FUNCTION_BLOCK "FB_SortingHeightAdvanced"   // FB18, SCL
{ S7_Optimized_Access := 'FALSE' }
VERSION : 0.4
// MANTIS â€” Scene 18: Sorting by Height (Advanced)  v0.4
//  Turntable-based 2-way sort: tall items â†’ LEFT, short â†’ RIGHT.
//  DB27, 76 bytes.  Enable flag at byte 74.
// 
//  I/O from Factory I/O driver (Siemens S7-1200/1500):
//    Inputs  %I0.0â€“%I1.7  (16 BOOLs)
//    Outputs %Q0.0â€“%Q1.4  (13 BOOLs) + %QD100 (DINT counter)
// 
//  Turntable notes:
//    Turn activates CW rotation; turntable snaps to 90Â° detents on stop.
//    AtFront = TRUE when turntable faces entry conveyor (0Â° position).
//    RIGHT exit â‰ˆ 90Â° CW from front  â†’ single turn, easy.
//    LEFT  exit â‰ˆ 270Â° CW from front â†’ timer-based (TURN_LEFT_TICKS).
//    Return to FRONT: Turn ON until AtFront = TRUE (always reliable).
//  ===== SENSORS (from Factory I/O) =====
   VAR
      AtEntry : Bool;   // %I0.0 Item at entry conveyor
      LowBox : Bool;   // %I0.1 Low height sensor triggered
      HighBox : Bool;   // %I0.2 High height sensor triggered
      AtTurntableEntry : Bool;   // %I0.3 Item at turntable entry area
      AtLoadPosition : Bool;   // %I0.4 Item centred on turntable
      AtUnloadPosition : Bool;   // %I0.5 Item at turntable unload edge
      AtFront : Bool;   // %I0.6 Turntable facing front (entry)
      AtRightEntry : Bool;   // %I0.7 Item entering right conveyor
      AtLeftEntry : Bool;   // %I1.0 Item entering left conveyor
      AtRightExit : Bool;   // %I1.1 Item at right conveyor exit
      AtLeftExit : Bool;   // %I1.2 Item at left conveyor exit
      BtnStart : Bool;   // %I1.3 Start button
      BtnReset : Bool;   // %I1.4 Reset button
      BtnStop : Bool;   // %I1.5 Stop button
      EmergencyStop : Bool;   // %I1.6 Emergency stop
      BtnAuto : Bool;   // %I1.7 Auto mode ===== ACTUATORS (to Factory I/O) =====
      FeederConveyor : Bool;   // %Q0.0 Feeder conveyor
      EntryConveyor : Bool;   // %Q0.1 Entry conveyor
      LoadAct : Bool;   // %Q0.2 Turntable rollers inward (load)
      UnloadAct : Bool;   // %Q0.3 Turntable rollers outward (unload)
      TurnAct : Bool;   // %Q0.4 Turntable rotate CW
      LeftConveyor : Bool;   // %Q0.5 Left exit conveyor
      RightConveyor : Bool;   // %Q0.6 Right exit conveyor
      GreenIndicator : Bool;   // %Q0.7 Green indicator
      YellowIndicator : Bool;   // %Q1.0 Yellow indicator
      RedIndicator : Bool;   // %Q1.1 Red indicator
      StartLight : Bool;   // %Q1.2 Start button light
      ResetLight : Bool;   // %Q1.3 Reset button light
      StopLight : Bool;   // %Q1.4 Stop button light
      CounterOut : DInt;   // (DINT) %QD100 Item counter display ===== INTERNAL =====
      iState : Int;   // State machine
      ItemCount : Int;   // Internal item counter
      IsTall : Bool;   // TRUE = tall (HighBox), FALSE = short
      TurnTimer : Int;   // Timer for LEFT 270Â° CW rotation
      DwellTimer : Int;   // General-purpose delay timer
      Running : Bool;   // System running flag
      Enable : Bool := TRUE;   // ATTACK SURFACE â€” PLC never writes
   END_VAR
BEGIN
       // ===== PANEL LIGHTS =====
       #StartLight := #Running;
       #ResetLight := NOT #Running;
       #StopLight := NOT #Running;

       // ===== INDICATORS =====
       #GreenIndicator := #Running AND (#iState >= 10);
       #YellowIndicator := #Running AND (#iState >= 40) AND (#iState <= 55);
       #RedIndicator := NOT #EmergencyStop OR NOT #Enable;

       // ===== COUNTER OUTPUT =====
       #CounterOut := INT_TO_DINT(#ItemCount);

       // ===== SAFETY / ENABLE CHECK =====
       IF NOT #EmergencyStop OR NOT #Enable THEN
           #FeederConveyor := FALSE;
           #EntryConveyor := FALSE;
           #LoadAct := FALSE;
           #UnloadAct := FALSE;
           #TurnAct := FALSE;
           #LeftConveyor := FALSE;
           #RightConveyor := FALSE;
           #Running := FALSE;
           #iState := 0;
           RETURN;
       END_IF;

       // ===== START / STOP / RESET =====
       IF #BtnStart AND NOT #Running AND #EmergencyStop THEN
           #Running := TRUE;
           #iState := 10;
       END_IF;

       IF NOT #BtnStop OR NOT #EmergencyStop THEN
           #Running := FALSE;
           #FeederConveyor := FALSE;
           #EntryConveyor := FALSE;
           #LoadAct := FALSE;
           #UnloadAct := FALSE;
           #TurnAct := FALSE;
           #LeftConveyor := FALSE;
           #RightConveyor := FALSE;
           #iState := 0;
       END_IF;

       IF #BtnReset THEN
           #ItemCount := 0;
           #IsTall := FALSE;
           #iState := 0;
           #Running := FALSE;
           #FeederConveyor := FALSE;
           #EntryConveyor := FALSE;
           #LoadAct := FALSE;
           #UnloadAct := FALSE;
           #TurnAct := FALSE;
           #LeftConveyor := FALSE;
           #RightConveyor := FALSE;
       END_IF;

       IF NOT #Running THEN
           #FeederConveyor := FALSE;
           #EntryConveyor := FALSE;
           #LoadAct := FALSE;
           #UnloadAct := FALSE;
           #TurnAct := FALSE;
           #LeftConveyor := FALSE;
           #RightConveyor := FALSE;
           RETURN;
       END_IF;

       // ===== EXIT CONVEYORS ALWAYS ON WHILE RUNNING =====
       #LeftConveyor := TRUE;
       #RightConveyor := TRUE;

       // ===== DEFAULT PROCESS OUTPUTS OFF (states set what they need) =====
       #FeederConveyor := FALSE;
       #EntryConveyor := FALSE;
       #LoadAct := FALSE;
       #UnloadAct := FALSE;
       #TurnAct := FALSE;

       // ===== STATE MACHINE =====
       CASE #iState OF

           0: // IDLE â€” waiting for start
               ;

               // ---------- FEED ----------
           10: // Run feeder + entry conveyors, detect height
               #FeederConveyor := TRUE;
               #EntryConveyor := TRUE;
               // Latch height while item passes sensors
               IF #HighBox THEN
                   #IsTall := TRUE;
               ELSIF #LowBox AND NOT #HighBox THEN
                   #IsTall := FALSE;
               END_IF;
               IF #AtTurntableEntry THEN
                   #iState := 20;
               END_IF;

               // ---------- LOAD ONTO TURNTABLE ----------
           20: // Turntable rollers pull item in
               #EntryConveyor := TRUE;
               #LoadAct := TRUE;
               IF #AtLoadPosition THEN
                   #DwellTimer := 0;
                   IF #IsTall THEN
                       #iState := 50;   // turn LEFT (270Â° CW)
                   ELSE
                       #iState := 40;   // turn RIGHT (90Â° CW)
                   END_IF;
               END_IF;

               // --------- TURN RIGHT  (90Â° CW from FRONT) ---------
           40: // Turn CW while still at FRONT; stop once we leave
               IF #AtFront THEN
                   #TurnAct := TRUE;
               ELSE
                   #DwellTimer := 0;
                   #iState := 45;
               END_IF;

           45: // Settle at RIGHT position
               #DwellTimer := #DwellTimer + 1;
               IF #DwellTimer >= 10 THEN
                   #DwellTimer := 0;
                   #iState := 60;
               END_IF;

               // --------- TURN LEFT  (270Â° CW from FRONT) ---------
               // Timer-based: ~30 ticks after leaving FRONT covers ~270Â°.
               // Calibrate if turntable speed differs from default.
           50: // Start turning CW, wait to leave FRONT
               #TurnAct := TRUE;
               IF NOT #AtFront THEN
                   #TurnTimer := 0;
                   #iState := 51;
               END_IF;

           51: // Keep turning CW past RIGHT and BACK toward LEFT
               #TurnAct := TRUE;
               #TurnTimer := #TurnTimer + 1;
               IF #TurnTimer >= 30 THEN
                   #DwellTimer := 0;
                   #iState := 55;
               END_IF;

           55: // Settle at LEFT position
               #DwellTimer := #DwellTimer + 1;
               IF #DwellTimer >= 10 THEN
                   #DwellTimer := 0;
                   #iState := 60;
               END_IF;

               // --------- UNLOAD ---------
           60: // Push item off turntable onto exit conveyor
               #UnloadAct := TRUE;
               #DwellTimer := #DwellTimer + 1;
               IF (#IsTall AND #AtLeftEntry) OR (NOT #IsTall AND #AtRightEntry)
                   OR (#DwellTimer >= 50) THEN
                   #DwellTimer := 0;
                   #iState := 70;
               END_IF;

               // --------- EXIT CONVEYOR ---------
           70: // Wait for item to reach exit sensor
               #DwellTimer := #DwellTimer + 1;
               IF (#IsTall AND #AtLeftExit) OR (NOT #IsTall AND #AtRightExit)
                   OR (#DwellTimer >= 50) THEN
                   #DwellTimer := 0;
                   #iState := 80;
               END_IF;

               // --------- RETURN TO FRONT ---------
           80: // Turn CW until AtFront
               #TurnAct := TRUE;
               IF #AtFront THEN
                   #DwellTimer := 0;
                   #iState := 85;
               END_IF;

           85: // Settle at FRONT
               #DwellTimer := #DwellTimer + 1;
               IF #DwellTimer >= 10 THEN
                   #iState := 90;
               END_IF;

               // --------- COUNT AND LOOP ---------
           90: // Increment counter, reset flags, loop
               #ItemCount := #ItemCount + 1;
               #IsTall := FALSE;
               #iState := 10;

       END_CASE;
END_FUNCTION_BLOCK

FUNCTION_BLOCK "FB_SortingHeightBasic"   // FB19, SCL
{ S7_Optimized_Access := 'FALSE' }
VERSION : 0.4
// MANTIS â€” Scene 19: Sorting by Height (Basic)
//  Sort items by height: short â†’ LEFT, tall â†’ RIGHT.
//  DB28: Instance DB (non-optimized access)
// 
//  Factory I/O layout:
//    Entry conveyor feeds items onto a pallet/loading area.
//    High sensor detects tall items. Low sensor detects short items.
//    Pallet sensor detects pallet ready. Loaded confirms item loaded.
//    Short box (Low sensor only) â†’ Transfer LEFT.
//    Tall  box (High sensor)     â†’ Transfer RIGHT.
//    Left and right exit conveyors carry sorted items away.
//    Start/Stop/Reset/EmergencyStop/Auto on control panel.
//    Counter display shows items sorted.
// 
//  Driver mapping (from Factory I/O):
//    SENSORS (Inputs):
//      NOTE: Use %I10.x/%I11.x (NOT %I0.x/%I1.x) because the PLC's
//      built-in physical DI module owns %IB0 and overwrites external writes.
//      High sensor      â†’ %I10.0
//      Low sensor       â†’ %I10.1
//      Pallet sensor    â†’ %I10.2
//      Loaded           â†’ %I10.3
//      At left entry    â†’ %I10.4
//      At left exit     â†’ %I10.5
//      At right entry   â†’ %I10.6
//      At right exit    â†’ %I10.7
//      Start            â†’ %I11.0
//      Reset            â†’ %I11.1
//      Stop             â†’ %I11.2
//      Emergency stop   â†’ %I11.3
//      Auto             â†’ %I11.4
//      FACTORY I/O (Running) â†’ %I11.5
// 
//    ACTUATORS (Outputs):
//      Conveyor entry   â†’ %Q0.0
//      Load             â†’ %Q0.1
//      Unload           â†’ %Q0.2
//      Transf. left     â†’ %Q0.3
//      Transf. right    â†’ %Q0.4
//      Conveyor left    â†’ %Q0.5
//      Conveyor right   â†’ %Q0.6
//      Start light      â†’ %Q0.7
//      Reset light      â†’ %Q1.0
//      Stop light       â†’ %Q1.1
//      Counter          â†’ (DINT) %QD100
// 
//  DB28 byte layout (non-optimized):
//    Sensors:
//      0:  HighSensor     2: LowSensor      4: PalletSensor
//      6:  Loaded         8: AtLeftEntry    10: AtLeftExit
//     12:  AtRightEntry  14: AtRightExit
//     16:  BtnStart      18: BtnReset      20: BtnStop
//     22:  EmergencyStop 24: BtnAuto
//    Actuators:
//     26:  ConveyorEntry 28: Load          30: Unload
//     32:  TransfLeft    34: TransfRight
//     36:  ConveyorLeft  38: ConveyorRight
//     40:  StartLight    42: ResetLight    44: StopLight
//     46-49: Counter (DINT)
//    Internal:
//     50:  iState (INT)    52: ItemCount (INT)
//     54:  IsTall (BOOL)   56: DwellTimer (INT)
//     58:  Running (BOOL)  60: Enable (BOOL)
//    Total = 62 bytes
// 
//  Sorting logic:
//    Low sensor ON only â†’ short item â†’ transfer LEFT
//    High sensor ON     â†’ tall item  â†’ transfer RIGHT
// 
//  Vulnerability: Enable (byte 60, default TRUE) â€” read but NEVER written.
//  â”€â”€ Sensors (inputs) â”€â”€
   VAR
      HighSensor : Bool;   // byte 0 â€” %I0.0
      _p00 : Byte;
      LowSensor : Bool;   // byte 2 â€” %I0.1
      _p01 : Byte;
      PalletSensor : Bool;   // byte 4 â€” %I0.2
      _p02 : Byte;
      Loaded : Bool;   // byte 6 â€” %I0.3
      _p03 : Byte;
      AtLeftEntry : Bool;   // byte 8 â€” %I0.4
      _p04 : Byte;
      AtLeftExit : Bool;   // byte 10 â€” %I0.5
      _p05 : Byte;
      AtRightEntry : Bool;   // byte 12 â€” %I0.6
      _p06 : Byte;
      AtRightExit : Bool;   // byte 14 â€” %I0.7
      _p07 : Byte;
      BtnStart : Bool;   // byte 16 â€” %I1.0
      _p08 : Byte;
      BtnReset : Bool;   // byte 18 â€” %I1.1
      _p09 : Byte;
      BtnStop : Bool;   // byte 20 â€” %I1.2
      _p10 : Byte;
      EmergencyStop : Bool;   // byte 22 â€” %I1.3
      _p11 : Byte;
      BtnAuto : Bool;   // byte 24 â€” %I1.4
      _p12 : Byte;   // â”€â”€ Actuators (outputs) â”€â”€
      ConveyorEntry : Bool;   // byte 26 â€” %Q0.0
      _p13 : Byte;
      LoadAct : Bool;   // byte 28 â€” %Q0.1 (Load)
      _p14 : Byte;
      UnloadAct : Bool;   // byte 30 â€” %Q0.2 (Unload)
      _p15 : Byte;
      TransfLeft : Bool;   // byte 32 â€” %Q0.3
      _p16 : Byte;
      TransfRight : Bool;   // byte 34 â€” %Q0.4
      _p17 : Byte;
      ConveyorLeft : Bool;   // byte 36 â€” %Q0.5
      _p18 : Byte;
      ConveyorRight : Bool;   // byte 38 â€” %Q0.6
      _p19 : Byte;
      StartLight : Bool;   // byte 40 â€” %Q0.7
      _p20 : Byte;
      ResetLight : Bool;   // byte 42 â€” %Q1.0
      _p21 : Byte;
      StopLight : Bool;   // byte 44 â€” %Q1.1
      _p22 : Byte;
      CounterOut : DInt := 0;   // byte 46 â€” %QD100 â”€â”€ Internal state â”€â”€
      iState : Int := 0;   // byte 50
      ItemCount : Int := 0;   // byte 52
      IsTall : Bool := FALSE;   // byte 54
      _p23 : Byte;
      DwellTimer : Int := 0;   // byte 56
      Running : Bool := FALSE;   // byte 58
      _p24 : Byte;
      Enable : Bool := TRUE;   // byte 60 â€” system enable (default ON)
      _p25 : Byte;   // Total: 62 bytes
   END_VAR
BEGIN
       // â•â•â•â•â•â•â•â•â•â•â•â•â•â•â•â•â•â•â•â•â•â•â•â•â•â•â•â•â•â•â•â•â•â•â•â•â•â•â•â•â•â•â•â•â•â•â•â•â•â•â•â•
       // Safety gate: if Enable is FALSE, shut everything down
       // â•â•â•â•â•â•â•â•â•â•â•â•â•â•â•â•â•â•â•â•â•â•â•â•â•â•â•â•â•â•â•â•â•â•â•â•â•â•â•â•â•â•â•â•â•â•â•â•â•â•â•â•
       IF NOT #Enable THEN
           #Running := FALSE;
           #ConveyorEntry := FALSE;
           #LoadAct := FALSE;
           #UnloadAct := FALSE;
           #TransfLeft := FALSE;
           #TransfRight := FALSE;
           #ConveyorLeft := FALSE;
           #ConveyorRight := FALSE;
           #StartLight := FALSE;
           #StopLight := TRUE;
           #ResetLight := FALSE;
           RETURN;
       END_IF;

       // â•â•â•â•â•â•â•â•â•â•â•â•â•â•â•â•â•â•â•â•â•â•â•â•â•â•â•â•â•â•â•â•â•â•â•â•â•â•â•â•â•â•â•â•â•â•â•â•â•â•â•â•
       // Button handling
       //
       // Factory I/O button types for this scene:
       //   Start  â†’ momentary, normally OPEN   (FALSE=idle, TRUE=pressed)
       //   Stop   â†’ momentary, normally CLOSED (TRUE=idle, FALSE=pressed)
       //   Reset  â†’ momentary, normally OPEN   (FALSE=idle, TRUE=pressed)
       //   E-Stop â†’ latching,  normally CLOSED (TRUE=normal, FALSE=engaged)
       //   Auto   â†’ selector switch
       // â•â•â•â•â•â•â•â•â•â•â•â•â•â•â•â•â•â•â•â•â•â•â•â•â•â•â•â•â•â•â•â•â•â•â•â•â•â•â•â•â•â•â•â•â•â•â•â•â•â•â•â•

       // Emergency stop is NC: FALSE when engaged â†’ stop
       IF NOT #EmergencyStop THEN
           #Running := FALSE;
       END_IF;

       // Stop is NC: FALSE when pressed â†’ stop
       IF NOT #BtnStop THEN
           #Running := FALSE;
       END_IF;

       // Start is NO: TRUE when pressed â†’ start (only if E-stop and Stop OK)
       IF #BtnStart AND NOT #Running AND #EmergencyStop AND #BtnStop THEN
           #Running := TRUE;
       END_IF;

       // Auto-start: if E-stop normal AND Stop not pressed, start automatically
       IF #EmergencyStop AND #BtnStop AND NOT #BtnStart THEN
           #Running := TRUE;
       END_IF;

       IF #BtnReset THEN
           #Running := FALSE;
           #iState := 0;
           #ItemCount := 0;
           #CounterOut := 0;
           #DwellTimer := 0;
           #IsTall := FALSE;
           #ConveyorEntry := FALSE;
           #LoadAct := FALSE;
           #UnloadAct := FALSE;
           #TransfLeft := FALSE;
           #TransfRight := FALSE;
           #ResetLight := TRUE;
           #StartLight := FALSE;
           #StopLight := FALSE;
           RETURN;
       END_IF;

       // â•â•â•â•â•â•â•â•â•â•â•â•â•â•â•â•â•â•â•â•â•â•â•â•â•â•â•â•â•â•â•â•â•â•â•â•â•â•â•â•â•â•â•â•â•â•â•â•â•â•â•â•
       // Panel indicator lights
       // â•â•â•â•â•â•â•â•â•â•â•â•â•â•â•â•â•â•â•â•â•â•â•â•â•â•â•â•â•â•â•â•â•â•â•â•â•â•â•â•â•â•â•â•â•â•â•â•â•â•â•â•
       #StartLight := #Running;
       #StopLight := NOT #Running;
       #ResetLight := FALSE;

       // â•â•â•â•â•â•â•â•â•â•â•â•â•â•â•â•â•â•â•â•â•â•â•â•â•â•â•â•â•â•â•â•â•â•â•â•â•â•â•â•â•â•â•â•â•â•â•â•â•â•â•â•
       // NOT running â†’ stop all actuators
       // â•â•â•â•â•â•â•â•â•â•â•â•â•â•â•â•â•â•â•â•â•â•â•â•â•â•â•â•â•â•â•â•â•â•â•â•â•â•â•â•â•â•â•â•â•â•â•â•â•â•â•â•
       IF NOT #Running THEN
           #ConveyorEntry := FALSE;
           #LoadAct := FALSE;
           #UnloadAct := FALSE;
           #TransfLeft := FALSE;
           #TransfRight := FALSE;
           #ConveyorLeft := FALSE;
           #ConveyorRight := FALSE;
           RETURN;
       END_IF;

       // â•â•â•â•â•â•â•â•â•â•â•â•â•â•â•â•â•â•â•â•â•â•â•â•â•â•â•â•â•â•â•â•â•â•â•â•â•â•â•â•â•â•â•â•â•â•â•â•â•â•â•â•
       // RUNNING â€” exit conveyors always ON
       // â•â•â•â•â•â•â•â•â•â•â•â•â•â•â•â•â•â•â•â•â•â•â•â•â•â•â•â•â•â•â•â•â•â•â•â•â•â•â•â•â•â•â•â•â•â•â•â•â•â•â•â•
       #ConveyorLeft := TRUE;
       #ConveyorRight := TRUE;

       // â•â•â•â•â•â•â•â•â•â•â•â•â•â•â•â•â•â•â•â•â•â•â•â•â•â•â•â•â•â•â•â•â•â•â•â•â•â•â•â•â•â•â•â•â•â•â•â•â•â•â•â•
       // Sorting state machine
       //   State 0: Feed â€” run entry conveyor, latch height, wait for pallet
       //   State 1: Load â€” lift transfer chains, wait for Loaded sensor
       //   State 2: Transfer â€” shortâ†’LEFT, tallâ†’RIGHT
       //   State 3: Clear â€” keep transfer ON while item clears center
       //   State 4: Finish â€” increment counter, return to feed
       //
       // Sorting direction:
       //   Low sensor only (short box)  â†’ Transfer LEFT
       //   High sensor (tall box)       â†’ Transfer RIGHT
       //
       // DwellTimer counts PLC scan cycles (~1-2 ms each on S7-1200).
       // Factory I/O mechanisms need real-world seconds, so thresholds
       // are in the thousands.
       // â•â•â•â•â•â•â•â•â•â•â•â•â•â•â•â•â•â•â•â•â•â•â•â•â•â•â•â•â•â•â•â•â•â•â•â•â•â•â•â•â•â•â•â•â•â•â•â•â•â•â•â•
       CASE #iState OF
           0: // â”€â”€ FEED: entry conveyor ON, detect height, wait for pallet â”€â”€
               #ConveyorEntry := TRUE;
               #LoadAct := FALSE;
               #UnloadAct := FALSE;
               #TransfLeft := FALSE;
               #TransfRight := FALSE;

               // Latch height sensors AS THE BOX APPROACHES on the entry conveyor.
               // The sensors fire as the box passes through â€” we must catch them
               // here in State 0 before the conveyor stops.
               IF #HighSensor THEN
                   #IsTall := TRUE;
               ELSIF #LowSensor THEN
                   #IsTall := FALSE;
               END_IF;

               IF #PalletSensor THEN
                   #DwellTimer := 0;
                   #iState := 1;
               END_IF;

           1: // â”€â”€ LOAD: run entry conveyor until box is fully loaded, then transfer â”€â”€
               // Entry conveyor keeps running until Loaded sensor fires
               // (box is fully on the loading platform and chains are raised).
               // Only then do we stop the conveyor and proceed to transfer.
               IF #Loaded THEN
                   #ConveyorEntry := FALSE;
               ELSE
                   #ConveyorEntry := TRUE;
               END_IF;
               #LoadAct := TRUE;         // Raise chains to lift box off rollers
               #UnloadAct := FALSE;
               #TransfLeft := FALSE;
               #TransfRight := FALSE;

               // Keep latching height sensors (they may still be active)
               IF #HighSensor THEN
                   #IsTall := TRUE;
               ELSIF #LowSensor THEN
                   #IsTall := FALSE;
               END_IF;

               #DwellTimer := #DwellTimer + 1;

               IF #Loaded THEN
                   // Box confirmed on platform â€” proceed to transfer
                   #DwellTimer := 0;
                   #iState := 2;
               ELSIF #DwellTimer > 5000 THEN
                   // Timeout (~5-10 s): Loaded never triggered, proceed anyway
                   #ConveyorEntry := FALSE;
                   #DwellTimer := 0;
                   #iState := 2;
               END_IF;

           2: // â”€â”€ TRANSFER: shortâ†’LEFT, tallâ†’RIGHT â”€â”€
               // Chains must stay raised (LoadAct=TRUE) while transfer runs.
               // Use TIMER ONLY â€” do NOT check AtLeftEntry/AtRightEntry because
               // those sensors may be permanently ON from previous boxes on the
               // exit conveyors.
               #ConveyorEntry := FALSE;
               #LoadAct := TRUE;         // KEEP chains raised during transfer!
               #UnloadAct := FALSE;

               IF #IsTall THEN
                   #TransfLeft := FALSE;
                   #TransfRight := TRUE;     // Tall â†’ RIGHT
               ELSE
                   #TransfLeft := TRUE;      // Short â†’ LEFT
                   #TransfRight := FALSE;
               END_IF;

               // Run transfer for a fixed duration (~5-10 seconds)
               #DwellTimer := #DwellTimer + 1;
               IF #DwellTimer > 5000 THEN
                   #iState := 3;
                   #DwellTimer := 0;
               END_IF;

           3: // â”€â”€ CLEAR: keep transfer ON so item fully clears center, then unload â”€â”€
               #ConveyorEntry := FALSE;

               IF #DwellTimer < 1500 THEN
                   // First ~1.5-3 s: keep chains UP + transfer running to push item off center
                   #LoadAct := TRUE;     // chains still raised
                   IF #IsTall THEN
                       #TransfLeft := FALSE;
                       #TransfRight := TRUE;
                   ELSE
                       #TransfLeft := TRUE;
                       #TransfRight := FALSE;
                   END_IF;
                   #UnloadAct := FALSE;
               ELSE
                   // Then: stop transfer, UNLOAD to lower chains back down
                   #LoadAct := FALSE;
                   #TransfLeft := FALSE;
                   #TransfRight := FALSE;
                   #UnloadAct := TRUE;
               END_IF;

               #DwellTimer := #DwellTimer + 1;
               IF #DwellTimer > 3000 THEN
                   // Total ~3-6 s dwell â€” item should be fully on exit conveyor
                   #iState := 4;
                   #DwellTimer := 0;
               END_IF;

           4: // â”€â”€ FINISH: count item, reset, return to feed â”€â”€
               #ConveyorEntry := FALSE;
               #LoadAct := FALSE;
               #UnloadAct := FALSE;
               #TransfLeft := FALSE;
               #TransfRight := FALSE;

               #ItemCount := #ItemCount + 1;
               #CounterOut := INT_TO_DINT(#ItemCount);
               #IsTall := FALSE;
               #iState := 0;

           ELSE
               // Unknown state â€” safe fallback
               #ConveyorEntry := FALSE;
               #LoadAct := FALSE;
               #UnloadAct := FALSE;
               #TransfLeft := FALSE;
               #TransfRight := FALSE;
               #iState := 0;
       END_CASE;
END_FUNCTION_BLOCK

FUNCTION_BLOCK "FB_SortingStation"   // FB20, SCL
{ S7_Optimized_Access := 'FALSE' }
VERSION : 0.1
// MANTIS â€” Scene 21: Sorting Station
//  Separate green and blue items using a vision sensor.
//  DB30: I/O mapping
   VAR
      ItemAtEntry : Bool;   // 0.0
      _pad0 : Byte;
      VisionColor : Int;   // 2 (0=none, 1=green, 2=blue)
      AtDiverter : Bool;   // 4.0
      _pad1 : Byte;
      AtExitGreen : Bool;   // 6.0
      _pad2 : Byte;
      AtExitBlue : Bool;   // 8.0
      _pad3 : Byte;
      ConveyorIn : Bool;   // 10.0
      _pad4 : Byte;
      ConveyorGreen : Bool;   // 12.0
      _pad5 : Byte;
      ConveyorBlue : Bool;   // 14.0
      _pad6 : Byte;
      Diverter : Bool;   // 16.0 (FALSE=green, TRUE=blue)
      _pad7 : Byte;
      Emitter : Bool;   // 18.0
      _pad8 : Byte;
      RemoverGreen : Bool;   // 20.0
      _pad9 : Byte;
      RemoverBlue : Bool;   // 22.0
      _pad10 : Byte;
      DetectedColor : Int := 0;
   END_VAR
BEGIN
       #Emitter := TRUE;
       #ConveyorIn := TRUE;
       #ConveyorGreen := TRUE;
       #ConveyorBlue := TRUE;
       #RemoverGreen := TRUE;
       #RemoverBlue := TRUE;

       // Detect color
       IF #ItemAtEntry AND #VisionColor > 0 THEN
           #DetectedColor := #VisionColor;
       END_IF;

       // Divert based on color
       IF #AtDiverter THEN
           IF #DetectedColor = 1 THEN
               #Diverter := FALSE;  // Green path
           ELSIF #DetectedColor = 2 THEN
               #Diverter := TRUE;   // Blue path
           END_IF;
       END_IF;
END_FUNCTION_BLOCK

FUNCTION_BLOCK "FB_SortingWeight"   // FB21, SCL
{ S7_Optimized_Access := 'FALSE' }
VERSION : 1.0
// MANTIS â€” Scene 20: Sorting by Weight
//  3-way weight sorter: weigh each box, then send left / forward / right.
//  DB22: Instance DB for FB_SortingWeight (non-optimized access)
// 
//  Factory I/O connections (ComDrvS7):
//    INPUTS (Bool Inputs Offset=10):
//      At scale entry  â†’ %I10.0      At forward entry â†’ %I10.5
//      At scale        â†’ %I10.1      At exit front    â†’ %I10.6
//      At scale exit   â†’ %I10.2      At right entry   â†’ %I10.7
//      At left entry   â†’ %I10.3      At exit right    â†’ %I11.0
//      At exit left    â†’ %I10.4      Start            â†’ %I11.1
//                                    Reset            â†’ %I11.2
//                                    Stop             â†’ %I11.3
//                                    Auto             â†’ %I11.4
//                                    FIO Running      â†’ %I11.5
//      Weight          â†’ %ID100 (REAL)
// 
//    OUTPUTS (Bool Outputs Offset=0):
//      Entry conveyor  â†’ %Q0.0       Front conveyor   â†’ %Q0.7
//      Load scale      â†’ %Q0.1       Start light      â†’ %Q1.0
//      Send left       â†’ %Q0.2       Reset light      â†’ %Q1.1
//      Left conveyor   â†’ %Q0.3       Stop light       â†’ %Q1.2
//      Send right      â†’ %Q0.4       Left count       â†’ %QD100 (DINT)
//      Right conveyor  â†’ %Q0.5       Forward count    â†’ %QD104 (DINT)
//      Send forward    â†’ %Q0.6       Right count      â†’ %QD108 (DINT)
//                                    Weight (display) â†’ %QD112 (DINT)
// 
//  DB22 byte layout (non-optimized):
//    -- Inputs --
//    Byte 0    : AtScaleEntry   (BOOL)
//    Byte 2    : AtScale        (BOOL)
//    Byte 4    : AtScaleExit    (BOOL)
//    Byte 6    : AtLeftEntry    (BOOL)
//    Byte 8    : AtExitLeft     (BOOL)
//    Byte 10   : AtForwardEntry (BOOL)
//    Byte 12   : AtExitFront    (BOOL)
//    Byte 14   : AtRightEntry   (BOOL)
//    Byte 16   : AtExitRight    (BOOL)
//    Byte 18   : BtnStart       (BOOL)
//    Byte 20   : BtnReset       (BOOL)
//    Byte 22   : BtnStop        (BOOL)
//    Byte 24   : BtnAuto        (BOOL)
//    Byte 26   : FIO_Running    (BOOL)
//    Byte 28   : Weight         (REAL)  â€” analog scale reading
//    -- Outputs --
//    Byte 32   : EntryConveyor  (BOOL)
//    Byte 34   : LoadScale      (BOOL)
//    Byte 36   : SendLeft       (BOOL)
//    Byte 38   : LeftConveyor   (BOOL)
//    Byte 40   : SendRight      (BOOL)
//    Byte 42   : RightConveyor  (BOOL)
//    Byte 44   : SendForward    (BOOL)
//    Byte 46   : FrontConveyor  (BOOL)
//    Byte 48   : StartLight     (BOOL)
//    Byte 50   : ResetLight     (BOOL)
//    Byte 52   : StopLight      (BOOL)
//    Byte 54   : LeftCount      (DINT)
//    Byte 58   : ForwardCount   (DINT)
//    Byte 62   : RightCount     (DINT)
//    Byte 66   : WeightDisplay  (DINT)
//    -- Internal --
//    Byte 70   : MeasuredWeight (REAL)
//    Byte 74   : LightThresh    (REAL)  â€” below = left
//    Byte 78   : HeavyThresh    (REAL)  â€” above = right, between = forward
//    Byte 82   : iState         (INT)
//    Byte 84   : Enable         (BOOL)
//    Total = 86 bytes
//  -- Inputs (sensors) --
   VAR
      AtScaleEntry : Bool;   // 0
      _p00 : Byte;
      AtScale : Bool;   // 2
      _p01 : Byte;
      AtScaleExit : Bool;   // 4
      _p02 : Byte;
      AtLeftEntry : Bool;   // 6
      _p03 : Byte;
      AtExitLeft : Bool;   // 8
      _p04 : Byte;
      AtForwardEntry : Bool;   // 10
      _p05 : Byte;
      AtExitFront : Bool;   // 12
      _p06 : Byte;
      AtRightEntry : Bool;   // 14
      _p07 : Byte;
      AtExitRight : Bool;   // 16
      _p08 : Byte;
      BtnStart : Bool;   // 18
      _p09 : Byte;
      BtnReset : Bool;   // 20
      _p10 : Byte;
      BtnStop : Bool;   // 22
      _p11 : Byte;
      BtnAuto : Bool;   // 24
      _p12 : Byte;
      FIO_Running : Bool;   // 26
      _p13 : Byte;
      Weight : Real;   // 28 â€” analog scale reading -- Outputs (actuators) --
      EntryConveyor : Bool;   // 32
      _p14 : Byte;
      LoadScale : Bool;   // 34
      _p15 : Byte;
      SendLeft : Bool;   // 36
      _p16 : Byte;
      LeftConveyor : Bool;   // 38
      _p17 : Byte;
      SendRight : Bool;   // 40
      _p18 : Byte;
      RightConveyor : Bool;   // 42
      _p19 : Byte;
      SendForward : Bool;   // 44
      _p20 : Byte;
      FrontConveyor : Bool;   // 46
      _p21 : Byte;
      StartLight : Bool;   // 48
      _p22 : Byte;
      ResetLight : Bool;   // 50
      _p23 : Byte;
      StopLight : Bool;   // 52
      _p24 : Byte;
      LeftCount : DInt;   // 54
      ForwardCount : DInt;   // 58
      RightCount : DInt;   // 62
      WeightDisplay : DInt;   // 66 -- Internal --
      MeasuredWeight : Real := 0.0;   // 70
      LightThresh : Real := 2.0;   // 74 â€” below this = light â†’ left
      HeavyThresh : Real := 5.0;   // 78 â€” above this = heavy â†’ right
      iState : Int := 0;   // 82
      Enable : Bool := TRUE;   // 84
      _p25 : Byte;   // 85 Total DB size: 86 bytes
   END_VAR
BEGIN
       // Exit conveyors always run to clear sorted boxes
       #LeftConveyor := TRUE;
       #FrontConveyor := TRUE;
       #RightConveyor := TRUE;

       // Lights mirror buttons
       #StartLight := #BtnStart OR #BtnAuto;
       #StopLight := #BtnStop;
       #ResetLight := #BtnReset;

       // Display current weight as integer (Ã—100 for display)
       #WeightDisplay := REAL_TO_DINT(#Weight * 100.0);

       // Default thresholds
       IF #LightThresh < 0.1 THEN
           #LightThresh := 2.0;
       END_IF;
       IF #HeavyThresh < 0.1 THEN
           #HeavyThresh := 5.0;
       END_IF;

       IF NOT #FIO_Running OR NOT #Enable THEN
           // Safe state
           #EntryConveyor := FALSE;
           #LoadScale := FALSE;
           #SendLeft := FALSE;
           #SendRight := FALSE;
           #SendForward := FALSE;
           #iState := 0;
       ELSE
           CASE #iState OF
               0: // Idle â€” feed box onto scale
                   #EntryConveyor := TRUE;
                   #LoadScale := TRUE;
                   #SendLeft := FALSE;
                   #SendRight := FALSE;
                   #SendForward := FALSE;
                   IF #AtScale THEN
                       // Box is on scale â€” stop to weigh
                       #EntryConveyor := FALSE;
                       #LoadScale := FALSE;
                       #MeasuredWeight := #Weight;
                       #iState := 1;
                   END_IF;

               1: // Weighed â€” decide direction
                   #EntryConveyor := FALSE;
                   #LoadScale := FALSE;
                   IF #MeasuredWeight < #LightThresh THEN
                       // Light â†’ send left
                       #SendLeft := TRUE;
                       #iState := 2;
                   ELSIF #MeasuredWeight >= #HeavyThresh THEN
                       // Heavy â†’ send right
                       #SendRight := TRUE;
                       #iState := 4;
                   ELSE
                       // Medium â†’ send forward
                       #SendForward := TRUE;
                       #iState := 6;
                   END_IF;

               2: // Sending left â€” wait for box to reach left entry
                   #SendLeft := TRUE;
                   #LoadScale := TRUE;  // run scale belt to push box off
                   IF #AtLeftEntry THEN
                       #SendLeft := FALSE;
                       #LoadScale := FALSE;
                       #LeftCount := #LeftCount + 1;
                       #iState := 0;
                   END_IF;

               3: // (unused â€” reserved)
                   #iState := 0;

               4: // Sending right â€” wait for box to reach right entry
                   #SendRight := TRUE;
                   #LoadScale := TRUE;
                   IF #AtRightEntry THEN
                       #SendRight := FALSE;
                       #LoadScale := FALSE;
                       #RightCount := #RightCount + 1;
                       #iState := 0;
                   END_IF;

               5: // (unused â€” reserved)
                   #iState := 0;

               6: // Sending forward â€” wait for box to reach forward entry
                   #SendForward := TRUE;
                   #LoadScale := TRUE;
                   IF #AtForwardEntry THEN
                       #SendForward := FALSE;
                       #LoadScale := FALSE;
                       #ForwardCount := #ForwardCount + 1;
                       #iState := 0;
                   END_IF;

               7: // (unused â€” reserved)
                   #iState := 0;
           END_CASE;
       END_IF;
END_FUNCTION_BLOCK

FUNCTION_BLOCK "FB_Warehouse"   // FB22, SCL
{ S7_Optimized_Access := 'FALSE' }
VERSION : 0.1
// MANTIS â€” Scene 7: Automated Warehouse
//  Transport, store and retrieve boxes from a rack using a stacker crane.
//  DB16: I/O mapping
   VAR
      AtEntry : Bool;   // 0.0
      _pad0 : Byte;
      AtExit : Bool;   // 2.0
      _pad1 : Byte;
      CraneX : Real;   // 4
      CraneZ : Real;   // 8
      CraneFork : Bool;   // 12.0
      _pad2 : Byte;
      ConveyorIn : Bool;   // 14.0
      _pad3 : Byte;
      ConveyorOut : Bool;   // 16.0
      _pad4 : Byte;
      CraneMoveX : Real;   // 18
      CraneMoveZ : Real;   // 22
      ForkExtend : Bool;   // 26.0
      _pad5 : Byte;
      ForkRetract : Bool;   // 28.0
      _pad6 : Byte;
      Emitter : Bool;   // 30.0
      _pad7 : Byte;
      TargetSlot : Int;   // 32
      iState : Int := 0;
      CurrentSlot : Int := 0;
      SLOT_SPACING_X : Real := 200.0;
      SLOT_SPACING_Z : Real := 150.0;
      COLS : Int := 5;
      TOLERANCE : Real := 15.0;
   END_VAR
BEGIN
       CASE #iState OF
           0: // Wait for box at entry
               #ConveyorIn := TRUE;
               #Emitter := TRUE;
               IF #AtEntry THEN
                   #ConveyorIn := FALSE;
                   #Emitter := FALSE;
                   // Calculate target position from slot
                   #CraneMoveX := INT_TO_REAL(#TargetSlot MOD #COLS) * #SLOT_SPACING_X;
                   #CraneMoveZ := INT_TO_REAL(#TargetSlot / #COLS) * #SLOT_SPACING_Z;
                   #iState := 1;
               END_IF;

           1: // Pick box at entry
               #ForkExtend := TRUE;
               IF #CraneFork THEN
                   #ForkExtend := FALSE;
                   #iState := 2;
               END_IF;

           2: // Move crane to target slot
               IF ABS(#CraneX - #CraneMoveX) < #TOLERANCE AND ABS(#CraneZ - #CraneMoveZ) < #TOLERANCE THEN
                   #iState := 3;
               END_IF;

           3: // Place box in slot
               #ForkRetract := TRUE;
               IF NOT #CraneFork THEN
                   #ForkRetract := FALSE;
                   // Move to next slot
                   #CurrentSlot := #CurrentSlot + 1;
                   IF #CurrentSlot > 24 THEN
                       #CurrentSlot := 0;
                   END_IF;
                   #TargetSlot := #CurrentSlot;
                   #CraneMoveX := 0.0;
                   #CraneMoveZ := 0.0;
                   #iState := 0;
               END_IF;
       END_CASE;
END_FUNCTION_BLOCK

ORGANIZATION_BLOCK "Main"   // OB1, SCL, ProgramCycle
{ S7_Optimized_Access := 'TRUE' }
VERSION : 0.1
// =============================================================================
//  MANTIS â€” TIA Portal Main Program (OB1)
//  
//  Calls the active scene's function block each scan cycle.
//  Set "ActiveScene" in DB1 to select which scene runs.
// 
//  Scene IDs:
//    1  = From A to B               (DB3)
//    2  = From A to B (Set/Reset)   (DB4)
//    3  = Filling Tank (Timers)     (DB5)
//    4  = Queue of Items (Counters) (DB6)
//    5  = Assembler                 (DB7)
//    6  = Assembler (Analog)        (DB8)
//    7  = Automated Warehouse       (DB9)
//    8  = Buffer Station            (DB10)
//    9  = Converge Station          (DB11)
//    10 = Elevator (Advanced)       (DB12)
//    11 = Elevator (Basic)          (DB13)
//    12 = Level Control             (DB14)
//    13 = Palletizer                (DB15)
//    14 = Pick & Place (Basic)      (DB16)
//    15 = Pick & Place XYZ          (DB17)
//    16 = Production Line           (DB18)
//    17 = Separating Station        (DB19)
//    18 = Sorting Height (Advanced) (DB20)
//    19 = Sorting Height (Basic)    (DB21)
//    20 = Sorting by Weight         (DB22)
//    21 = Sorting Station           (DB23)
//  =============================================================================
   VAR_INPUT
      Initial_Call : Bool;   // Initial call of this OB
      Remanence : Bool;   // =True, if remanent data are available
   END_VAR
BEGIN
       // Call the active scene FB based on DB1.ActiveScene
       // Each scene uses its own instance DB

       // ================================================================
       // I/O BRIDGE â€” Maps Factory I/O %I/%Q to Scene DB variables.
       //
       // Factory I/O communicates via physical I/O addresses (%I, %Q).
       // MANTIS reads/writes via Data Blocks (DB) using Snap7.
       // This bridge copies:
       //   %I (sensors)   â†’ DB  (before FB call)
       //   DB (actuators) â†’ %Q  (after FB call)
       //
       // I/O assignment rule:
       //   BOOL sensors:   %I10.0, %I10.1, ... (offset 10 â€” avoids S7-1200 built-in DI at %IB0)
       //   BOOL actuators: %Q0.0,  %Q0.1,  ... (sequential bits, no conflict)
       //   DWORD inputs:   %ID100, %ID104, ...
       //   DWORD outputs:  %QD100, %QD104, ...
       //
       // IMPORTANT: The S7-1200 CPU has a built-in physical digital input module
       // at %I0.0-%I0.7 (and possibly %I1.x). The PLC overwrites these from the
       // hardware pins every scan cycle, so Factory I/O PUT/GET writes to %I0.x
       // are immediately lost. ALL sensor inputs are therefore mapped to %I10.x+
       // where no physical module exists, allowing Factory I/O writes to persist.
       //
       // In the Factory I/O S7 COMM driver, set Bool Inputs Offset = 10.
       // ================================================================

       // â”€â”€ Clear ALL outputs before scene-specific writes â”€â”€
       // Prevents stale bits from a previously-active scene confusing Factory I/O.
       "Tag__639094559022291825" := 0;
       "Tag__639094559022387271" := 0;
       "Tag__639094559022442425" := 0;
       "Tag__639094559022502581" := 0;
       "Tag__639094376040963045" := 0;
       "Tag__639094376042315926" := 0;
       "Tag__639094376042397245" := 0;
       "Tag__639094376042397246" := 0;

       CASE "DB_Config".ActiveScene OF

           1:  // Scene 1: From A to B (DB3)
               // Sensors: 1 BOOL â€” remapped to %I10.x (avoid built-in DI module)
               "FB_FromAtoB_DB".Sensor := "Tag__639094376038885860";
               // Run FB
               "FB_FromAtoB_DB"();
               // Actuators: 1 BOOL (conveyor only, emitter/remover are automatic)
               "Tag__639094376037924724" := "FB_FromAtoB_DB".Conveyor;

           2:  // Scene 2: From A to B Set/Reset (DB4)
               // 3 Bool inputs remapped to %I10.x
               "FB_FromAtoB_SR_DB".SensorA := "Tag__639094376038885860";
               "FB_FromAtoB_SR_DB".SensorB := "Tag__639094376038885861";
               "FB_FromAtoB_SR_DB".FIO_Running := "Tag__639094376039046363";
               // Run FB
               "FB_FromAtoB_SR_DB"();
               // 1 Bool output: Conveyor=%Q0.0
               "Tag__639094376037924724" := "FB_FromAtoB_SR_DB".Conveyor;

           3:  // Scene 3: Filling Tank (DB5)
               // 3 Bool inputs: Fill=%I10.0, Discharge=%I10.1, FIO_Running=%I10.2
               "FB_FillingTank_DB".SensorFill := "Tag__639094376038885860";
               "FB_FillingTank_DB".SensorDrain := "Tag__639094376038885861";
               "FB_FillingTank_DB".FIO_Running := "Tag__639094376039046363";
               "FB_FillingTank_DB"();
               // 4 Bool outputs: FillValve=%Q0.0, Filling=%Q0.1, DrainValve=%Q0.2, Discharging=%Q0.3
               "Tag__639094376037924724" := "FB_FillingTank_DB".FillValve;
               "Tag__639094376038085904" := "FB_FillingTank_DB".Filling;
               "Tag__639094376038085905" := "FB_FillingTank_DB".DrainValve;
               "Tag__639094376038405653" := "FB_FillingTank_DB".Discharging;

           4:  // Scene 4: Queue of Items (DB6)
               // Sensors â€” remapped to %I10.x (avoid built-in DI module)
               "FB_QueueItems_DB".AtEntry := "Tag__639094376038885860";
               "FB_QueueItems_DB".AtExit := "Tag__639094376038885861";
               "FB_QueueItems_DB"();
               "Tag__639094376037924724" := "FB_QueueItems_DB".Conveyor;
               "Tag__639094376038085904" := "FB_QueueItems_DB".Emitter;
               "Tag__639094376038085905" := "FB_QueueItems_DB".Remover;

           5:  // Scene 5: Assembler (DB7)
               // Sensors â€” remapped to %I10.x (avoid built-in DI module)
               "FB_Assembler_DB".PartAtPickup := "Tag__639094376038885860";
               "FB_Assembler_DB".PartAtPlace := "Tag__639094376038885861";
               "FB_Assembler_DB".LidAtPickup := "Tag__639094376039046363";
               "FB_Assembler_DB".ClampSensor := "Tag__639094376039046364";
               "FB_Assembler_DB".MovingX := "Tag__639094376039046365";
               "FB_Assembler_DB".MovingZ := "Tag__639094376039205258";
               "FB_Assembler_DB"();
               "Tag__639094376037924724" := "FB_Assembler_DB".ConveyorBase;
               "Tag__639094376038085904" := "FB_Assembler_DB".ConveyorLid;
               "Tag__639094376038085905" := "FB_Assembler_DB".ConveyorOut;
               "Tag__639094376038405653" := "FB_Assembler_DB".MoveX;
               "Tag__639094376038565707" := "FB_Assembler_DB".MoveZ;
               "Tag__639094376038565708" := "FB_Assembler_DB".Clamp;
               "Tag__639094376038565709" := "FB_Assembler_DB".Emitter;

           6:  // Scene 6: Assembler Analog (DB8) â€” has REAL I/O
               // Sensors â€” remapped to %I10.x (avoid built-in DI module)
               "FB_AssemblerAnalog_DB".PartAtPickup := "Tag__639094376038885860";
               "FB_AssemblerAnalog_DB".PartAtPlace := "Tag__639094376038885861";
               "FB_AssemblerAnalog_DB".LidAtPickup := "Tag__639094376039046363";
               "FB_AssemblerAnalog_DB".ClampSensor := "Tag__639094376039046364";
               "FB_AssemblerAnalog_DB"();
               "Tag__639094376037924724" := "FB_AssemblerAnalog_DB".ConveyorBase;
               "Tag__639094376038085904" := "FB_AssemblerAnalog_DB".ConveyorLid;
               "Tag__639094376038085905" := "FB_AssemblerAnalog_DB".ConveyorOut;
               "Tag__639094376038405653" := "FB_AssemblerAnalog_DB".Clamp;
               "Tag__639094376038565707" := "FB_AssemblerAnalog_DB".Emitter;
               // NOTE: REAL I/O (PosX, PosZ, SetpointX, SetpointZ) need
               // analog mapping â€” configure in Factory I/O driver.

           7:  // Scene 7: Automated Warehouse (DB9)
               // Sensors â€” remapped to %I10.x (avoid built-in DI module)
               "FB_Warehouse_DB".AtEntry := "Tag__639094376038885860";
               "FB_Warehouse_DB".AtExit := "Tag__639094376038885861";
               "FB_Warehouse_DB".CraneFork := "Tag__639094376039046363";
               "FB_Warehouse_DB"();
               "Tag__639094376037924724" := "FB_Warehouse_DB".ConveyorIn;
               "Tag__639094376038085904" := "FB_Warehouse_DB".ConveyorOut;
               "Tag__639094376038085905" := "FB_Warehouse_DB".ForkExtend;
               "Tag__639094376038405653" := "FB_Warehouse_DB".ForkRetract;
               "Tag__639094376038565707" := "FB_Warehouse_DB".Emitter;
               // NOTE: REAL I/O (CraneX, CraneZ, CraneMoveX, CraneMoveZ) need
               // analog mapping â€” configure in Factory I/O driver.

           8:  // Scene 8: Buffer Station (DB10)
               // Sensors â€” remapped to %I10.x (avoid built-in DI module)
               "FB_BufferStation_DB".Sensor1 := "Tag__639094376038885860";
               "FB_BufferStation_DB".Sensor2 := "Tag__639094376038885861";
               "FB_BufferStation_DB".Sensor3 := "Tag__639094376039046363";
               "FB_BufferStation_DB".Sensor4 := "Tag__639094376039046364";
               "FB_BufferStation_DB".Sensor5 := "Tag__639094376039046365";
               "FB_BufferStation_DB".AtExit := "Tag__639094376039205258";
               "FB_BufferStation_DB"();
               "Tag__639094376037924724" := "FB_BufferStation_DB".Conveyor;
               "Tag__639094376038085904" := "FB_BufferStation_DB".Stopper1;
               "Tag__639094376038085905" := "FB_BufferStation_DB".Stopper2;
               "Tag__639094376038405653" := "FB_BufferStation_DB".Emitter;
               "Tag__639094376038565707" := "FB_BufferStation_DB".Remover;

           9:  // Scene 9: Converge Station (DB11)
               // Sensors â€” remapped to %I10.x (avoid built-in DI module)
               "FB_ConvergeStation_DB".SensorLeft := "Tag__639094376038885860";
               "FB_ConvergeStation_DB".SensorRight := "Tag__639094376038885861";
               "FB_ConvergeStation_DB".SensorMerge := "Tag__639094376039046363";
               "FB_ConvergeStation_DB".AtExit := "Tag__639094376039046364";
               "FB_ConvergeStation_DB"();
               "Tag__639094376037924724" := "FB_ConvergeStation_DB".ConveyorLeft;
               "Tag__639094376038085904" := "FB_ConvergeStation_DB".ConveyorRight;
               "Tag__639094376038085905" := "FB_ConvergeStation_DB".ConveyorOut;
               "Tag__639094376038405653" := "FB_ConvergeStation_DB".Emitter1;
               "Tag__639094376038565707" := "FB_ConvergeStation_DB".Emitter2;
               "Tag__639094376038565708" := "FB_ConvergeStation_DB".Remover;

           10: // Scene 10: Elevator Advanced (DB12) â€” 20 inputs, 26 BOOL + 1 DINT outputs
               // â”€â”€ Sensors (inputs) â”€â”€ NOTE: remapped to %I10.x+ to avoid built-in DI conflict
               "FB_ElevatorAdvanced_DB".At1 := "Tag__639094376038885860";
               "FB_ElevatorAdvanced_DB".At2 := "Tag__639094376038885861";
               "FB_ElevatorAdvanced_DB".At3 := "Tag__639094376039046363";
               "FB_ElevatorAdvanced_DB".AtElevator := "Tag__639094376039046364";
               "FB_ElevatorAdvanced_DB".AtEntry := "Tag__639094376039046365";
               "FB_ElevatorAdvanced_DB".AtExit := "Tag__639094376039205258";
               "FB_ElevatorAdvanced_DB".At0Low := "Tag__639094376039205259";
               "FB_ElevatorAdvanced_DB".At0High := "Tag__639094376039205260";
               "FB_ElevatorAdvanced_DB".At1Low := "Tag__639094376039365268";
               "FB_ElevatorAdvanced_DB".At1High := "Tag__639094376039365269";
               "FB_ElevatorAdvanced_DB".At2Low := "Tag__639094376039365270";
               "FB_ElevatorAdvanced_DB".At2High := "Tag__639094376039525211";
               "FB_ElevatorAdvanced_DB".At3Low := "Tag__639094376039525212";
               "FB_ElevatorAdvanced_DB".At3High := "Tag__639094376039525213";
               "FB_ElevatorAdvanced_DB".BtnStart := "Tag__639094376039685481";
               "FB_ElevatorAdvanced_DB".BtnReset := "Tag__639094376039685482";
               "FB_ElevatorAdvanced_DB".BtnStop := "Tag__639094376039685483";
               "FB_ElevatorAdvanced_DB".EmergencyStop := "Tag__639094376039846408";
               "FB_ElevatorAdvanced_DB".BtnAuto := "Tag__639094376039846409";

               "FB_ElevatorAdvanced_DB"();

               // â”€â”€ Actuators (outputs) â”€â”€
               "Tag__639094376037924724" := "FB_ElevatorAdvanced_DB".Conveyor0;
               "Tag__639094376038085904" := "FB_ElevatorAdvanced_DB".Conveyor1;
               "Tag__639094376038085905" := "FB_ElevatorAdvanced_DB".Conveyor2;
               "Tag__639094376038405653" := "FB_ElevatorAdvanced_DB".Conveyor3;
               "Tag__639094376038565707" := "FB_ElevatorAdvanced_DB".ExitConveyor;
               "Tag__639094376038565708" := "FB_ElevatorAdvanced_DB".Load;
               "Tag__639094376039846410" := "FB_ElevatorAdvanced_DB".Unload;
               "Tag__639094376040005546" := "FB_ElevatorAdvanced_DB".Up;
               "Tag__639094376038565709" := "FB_ElevatorAdvanced_DB".Down;
               "Tag__639094376040005547" := "FB_ElevatorAdvanced_DB".Slow;
               "Tag__639094376040005548" := "FB_ElevatorAdvanced_DB".WarningLight;
               "Tag__639094376040163908" := "FB_ElevatorAdvanced_DB".StartLight;
               "Tag__639094376040163909" := "FB_ElevatorAdvanced_DB".ResetLight;
               "Tag__639094376040163910" := "FB_ElevatorAdvanced_DB".StopLight;
               "Tag__639094376040323143" := "FB_ElevatorAdvanced_DB".Floor1Ind;
               "Tag__639094376040323144" := "FB_ElevatorAdvanced_DB".Floor2Ind;
               "Tag__639094376040323145" := "FB_ElevatorAdvanced_DB".Floor3Ind;
               "Tag__639094376040483081" := "FB_ElevatorAdvanced_DB".Green1;
               "Tag__639094376040483082" := "FB_ElevatorAdvanced_DB".Yellow1;
               "Tag__639094376040483083" := "FB_ElevatorAdvanced_DB".Red1;
               "Tag__639094376040642647" := "FB_ElevatorAdvanced_DB".Green2;
               "Tag__639094376040642648" := "FB_ElevatorAdvanced_DB".Yellow2;
               "Tag__639094376040642649" := "FB_ElevatorAdvanced_DB".Red2;
               "Tag__639094376040802767" := "FB_ElevatorAdvanced_DB".Green3;
               "Tag__639094376040802768" := "FB_ElevatorAdvanced_DB".Yellow3;
               "Tag__639094376040802769" := "FB_ElevatorAdvanced_DB".Red3;
               // DINT output for display
               "Tag__639094376040963045" := DINT_TO_DWORD("FB_ElevatorAdvanced_DB".Display);

           11: // Scene 11: Elevator Basic (DB13) â€” 30 inputs, 29 outputs
               // â”€â”€ Sensors (inputs) â”€â”€
               // NOTE: Use %I10.x-%I13.x to avoid built-in DI module conflict
               "FB_ElevatorBasic_DB".AtEntry := "Tag__639094376038885860";
               "FB_ElevatorBasic_DB".AtEntryLeft := "Tag__639094376038885861";
               "FB_ElevatorBasic_DB".AtExitLeft := "Tag__639094376039046363";
               "FB_ElevatorBasic_DB".AtEntry0 := "Tag__639094376039046364";
               "FB_ElevatorBasic_DB".AtExit0 := "Tag__639094376039046365";
               "FB_ElevatorBasic_DB".AtEntryRight := "Tag__639094376039205258";
               "FB_ElevatorBasic_DB".AtExitRight := "Tag__639094376039205259";
               "FB_ElevatorBasic_DB".AtExit := "Tag__639094376039205260";
               "FB_ElevatorBasic_DB".AtEntry1 := "Tag__639094376039365268";
               "FB_ElevatorBasic_DB".AtExit1 := "Tag__639094376039365269";
               "FB_ElevatorBasic_DB".AtEntry2 := "Tag__639094376039365270";
               "FB_ElevatorBasic_DB".AtExit2 := "Tag__639094376039525211";
               "FB_ElevatorBasic_DB".AtLeftLow0 := "Tag__639094376039525212";
               "FB_ElevatorBasic_DB".AtLeftHigh0 := "Tag__639094376039525213";
               "FB_ElevatorBasic_DB".AtLeftLow1 := "Tag__639094376039685481";
               "FB_ElevatorBasic_DB".AtLeftHigh1 := "Tag__639094376039685482";
               "FB_ElevatorBasic_DB".AtLeftLow2 := "Tag__639094376039685483";
               "FB_ElevatorBasic_DB".AtLeftHigh2 := "Tag__639094376039846408";
               "FB_ElevatorBasic_DB".AtRightLow0 := "Tag__639094376039846409";
               "FB_ElevatorBasic_DB".AtRightHigh0 := "Tag__639094376041124518";
               "FB_ElevatorBasic_DB".AtRightLow1 := "Tag__639094376041124519";
               "FB_ElevatorBasic_DB".AtRightHigh1 := "Tag__639094376041283188";
               "FB_ElevatorBasic_DB".AtRightLow2 := "Tag__639094376041283189";
               "FB_ElevatorBasic_DB".AtRightHigh2 := "Tag__639094376041283190";
               "FB_ElevatorBasic_DB".BtnStart := "Tag__639094376041442043";
               "FB_ElevatorBasic_DB".BtnReset := "Tag__639094376041442044";
               "FB_ElevatorBasic_DB".BtnStop := "Tag__639094376041600752";
               "FB_ElevatorBasic_DB".EmergencyStop := "Tag__639094376041600753";
               "FB_ElevatorBasic_DB".BtnAuto := "Tag__639094376041600754";

               "FB_ElevatorBasic_DB"();

               // â”€â”€ Actuators (outputs) â”€â”€
               "Tag__639094376037924724" := "FB_ElevatorBasic_DB".EntryConveyor;
               "Tag__639094376038085904" := "FB_ElevatorBasic_DB".UnloadLeft;
               "Tag__639094376038085905" := "FB_ElevatorBasic_DB".LoadLeft;
               "Tag__639094376038405653" := "FB_ElevatorBasic_DB".Conveyor0;
               "Tag__639094376038565707" := "FB_ElevatorBasic_DB".UnloadRight;
               "Tag__639094376038565708" := "FB_ElevatorBasic_DB".LoadRight;
               "Tag__639094376039846410" := "FB_ElevatorBasic_DB".ExitConveyor;
               "Tag__639094376040005546" := "FB_ElevatorBasic_DB".LeftUp;
               "Tag__639094376038565709" := "FB_ElevatorBasic_DB".LeftSlow;
               "Tag__639094376040005547" := "FB_ElevatorBasic_DB".LeftDown;
               "Tag__639094376040005548" := "FB_ElevatorBasic_DB".RightUp;
               "Tag__639094376040163908" := "FB_ElevatorBasic_DB".RightSlow;
               "Tag__639094376040163909" := "FB_ElevatorBasic_DB".RightDown;
               "Tag__639094376040163910" := "FB_ElevatorBasic_DB".Conveyor1;
               "Tag__639094376040323143" := "FB_ElevatorBasic_DB".Conveyor2;
               "Tag__639094376040323144" := "FB_ElevatorBasic_DB".LeftWarning;
               "Tag__639094376040323145" := "FB_ElevatorBasic_DB".RightWarning;
               "Tag__639094376040483081" := "FB_ElevatorBasic_DB".Green0;
               "Tag__639094376040483082" := "FB_ElevatorBasic_DB".Yellow0;
               "Tag__639094376040483083" := "FB_ElevatorBasic_DB".Red0;
               "Tag__639094376040642647" := "FB_ElevatorBasic_DB".BGreen;
               "Tag__639094376040642648" := "FB_ElevatorBasic_DB".BYellow;
               "Tag__639094376040642649" := "FB_ElevatorBasic_DB".BRed;
               "Tag__639094376040802767" := "FB_ElevatorBasic_DB".CGreen;
               "Tag__639094376040802768" := "FB_ElevatorBasic_DB".CYellow;
               "Tag__639094376040802769" := "FB_ElevatorBasic_DB".CRed;
               "Tag__639094376041760860" := "FB_ElevatorBasic_DB".StartLight;
               "Tag__639094376041918319" := "FB_ElevatorBasic_DB".ResetLight;
               "Tag__639094376041918320" := "FB_ElevatorBasic_DB".StopLight;

           12: // Scene 12: Level Control (DB14) â€” BOOL + analog REAL/DINT I/O
               // BOOL inputs â€” use %I10.x to avoid built-in DI module conflict
               "FB_LevelControl_DB".Start := "Tag__639094376038885860";
               "FB_LevelControl_DB".Reset := "Tag__639094376038885861";
               "FB_LevelControl_DB".Stop := "Tag__639094376039046363";
               // Analog inputs (REAL via DWORD reinterpret)
               "FB_LevelControl_DB".LevelMeter := DWORD_TO_REAL("Tag__639094376042076147");
               "FB_LevelControl_DB".FlowMeter := DWORD_TO_REAL("Tag__639094376042076148");
               // Setpoint knob: copy ONLY while system is stopped.
               // Once Running=TRUE, SetpointIn freezes â†’ becomes write-once attack target.
               IF NOT "FB_LevelControl_DB".Running THEN
                   "FB_LevelControl_DB".SetpointIn := DWORD_TO_REAL("Tag__639094376042235578");
               END_IF;

               "FB_LevelControl_DB"();

               // BOOL outputs
               "Tag__639094376037924724" := "FB_LevelControl_DB".StartLight;
               "Tag__639094376038085904" := "FB_LevelControl_DB".ResetLight;
               "Tag__639094376038085905" := "FB_LevelControl_DB".StopLight;
               // Analog outputs (REAL via DWORD reinterpret)
               "Tag__639094376040963045" := REAL_TO_DWORD("FB_LevelControl_DB".FillValve);
               "Tag__639094376042315926" := REAL_TO_DWORD("FB_LevelControl_DB".DischargeValve);
               // DINT outputs for SP/PV displays
               "Tag__639094376042397245" := DINT_TO_DWORD("FB_LevelControl_DB".SP_Display);
               "Tag__639094376042397246" := DINT_TO_DWORD("FB_LevelControl_DB".PV_Display);

           13: // Scene 13: Palletizer (DB15)
               // Sensors â€” remapped to %I10.x (avoid built-in DI module)
               "FB_Palletizer_DB".BoxAtEntry := "Tag__639094376038885860";
               "FB_Palletizer_DB".BoxAtPickup := "Tag__639094376038885861";
               "FB_Palletizer_DB".PalletReady := "Tag__639094376039046363";
               "FB_Palletizer_DB".LayerComplete := "Tag__639094376039046364";
               "FB_Palletizer_DB".ClampSensor := "Tag__639094376039046365";
               "FB_Palletizer_DB"();
               "Tag__639094376037924724" := "FB_Palletizer_DB".ConveyorIn;
               "Tag__639094376038085904" := "FB_Palletizer_DB".Clamp;
               "Tag__639094376038085905" := "FB_Palletizer_DB".ConveyorOut;
               "Tag__639094376038405653" := "FB_Palletizer_DB".Emitter;
               // NOTE: REAL I/O (PosX, PosZ, MoveX, MoveZ) need analog mapping.

           14: // Scene 14: Pick & Place Basic (DB16)
               // Sensors â€” remapped to %I10.x (avoid built-in DI module)
               "FB_PickPlaceBasic_DB".ItemAtPick := "Tag__639094376038885860";
               "FB_PickPlaceBasic_DB".ItemAtPlace := "Tag__639094376038885861";
               "FB_PickPlaceBasic_DB".GripperClosed := "Tag__639094376039046363";
               "FB_PickPlaceBasic_DB".ArmAtPick := "Tag__639094376039046364";
               "FB_PickPlaceBasic_DB".ArmAtPlace := "Tag__639094376039046365";
               "FB_PickPlaceBasic_DB"();
               "Tag__639094376037924724" := "FB_PickPlaceBasic_DB".ConveyorIn;
               "Tag__639094376038085904" := "FB_PickPlaceBasic_DB".ConveyorOut;
               "Tag__639094376038085905" := "FB_PickPlaceBasic_DB".Gripper;
               "Tag__639094376038405653" := "FB_PickPlaceBasic_DB".ArmRotate;
               "Tag__639094376038565707" := "FB_PickPlaceBasic_DB".ArmUp;
               "Tag__639094376038565708" := "FB_PickPlaceBasic_DB".ArmDown;
               "Tag__639094376038565709" := "FB_PickPlaceBasic_DB".Emitter;

           15: // Scene 15: Pick & Place XYZ (DB17)
               // Sensors â€” remapped to %I10.x (avoid built-in DI module)
               "FB_PickPlaceXYZ_DB".BoxAtPick := "Tag__639094376038885860";
               "FB_PickPlaceXYZ_DB".PalletReady := "Tag__639094376038885861";
               "FB_PickPlaceXYZ_DB".GripperClosed := "Tag__639094376039046363";
               "FB_PickPlaceXYZ_DB"();
               "Tag__639094376037924724" := "FB_PickPlaceXYZ_DB".Gripper;
               "Tag__639094376038085904" := "FB_PickPlaceXYZ_DB".ConveyorIn;
               "Tag__639094376038085905" := "FB_PickPlaceXYZ_DB".ConveyorPallet;
               "Tag__639094376038405653" := "FB_PickPlaceXYZ_DB".Emitter;
               // NOTE: REAL I/O (PosX, PosY, PosZ, SetpointX, SetpointY, SetpointZ)
               // need analog mapping â€” configure in Factory I/O driver.

           16: // Scene 16: Production Line (DB18)
               // Sensors â€” remapped to %I10.x (avoid built-in DI module)
               "FB_ProductionLine_DB".LidReady := "Tag__639094376038885860";
               "FB_ProductionLine_DB".BaseReady := "Tag__639094376038885861";
               "FB_ProductionLine_DB".LidAtAssembly := "Tag__639094376039046363";
               "FB_ProductionLine_DB".BaseAtAssembly := "Tag__639094376039046364";
               "FB_ProductionLine_DB"();
               "Tag__639094376037924724" := "FB_ProductionLine_DB".LidMachine;
               "Tag__639094376038085904" := "FB_ProductionLine_DB".BaseMachine;
               "Tag__639094376038085905" := "FB_ProductionLine_DB".ConveyorLid;
               "Tag__639094376038405653" := "FB_ProductionLine_DB".ConveyorBase;
               "Tag__639094376038565707" := "FB_ProductionLine_DB".ConveyorOut;
               "Tag__639094376038565708" := "FB_ProductionLine_DB".Emitter;
               // NOTE: INT I/O (LidCount, BaseCount) need word mapping.

           17: // Scene 17: Separating Station (DB19)
               // Sensors â€” remapped to %I10.x (avoid built-in DI module)
               "FB_SeparatingStation_DB".PartAtEntry := "Tag__639094376038885860";
               "FB_SeparatingStation_DB".AtDiverter := "Tag__639094376038885861";
               "FB_SeparatingStation_DB".AtExitLeft := "Tag__639094376039046363";
               "FB_SeparatingStation_DB".AtExitRight := "Tag__639094376039046364";
               "FB_SeparatingStation_DB"();
               "Tag__639094376037924724" := "FB_SeparatingStation_DB".ConveyorIn;
               "Tag__639094376038085904" := "FB_SeparatingStation_DB".ConveyorLeft;
               "Tag__639094376038085905" := "FB_SeparatingStation_DB".ConveyorRight;
               "Tag__639094376038405653" := "FB_SeparatingStation_DB".Diverter;
               "Tag__639094376038565707" := "FB_SeparatingStation_DB".Emitter;
               "Tag__639094376038565708" := "FB_SeparatingStation_DB".RemoverLeft;
               "Tag__639094376038565709" := "FB_SeparatingStation_DB".RemoverRight;
               // NOTE: INT I/O (VisionSensor) needs word mapping.

           18: // Scene 18: Sorting Height Advanced (DB20) â€” 16 inputs, 13 BOOL + 1 DINT outputs
               // â”€â”€ Sensors (inputs) â€” remapped to %I10.x/%I11.x (avoid built-in DI module) â”€â”€
               "FB_SortingHeightAdv_DB".AtEntry := "Tag__639094376038885860";
               "FB_SortingHeightAdv_DB".LowBox := "Tag__639094376038885861";
               "FB_SortingHeightAdv_DB".HighBox := "Tag__639094376039046363";
               "FB_SortingHeightAdv_DB".AtTurntableEntry := "Tag__639094376039046364";
               "FB_SortingHeightAdv_DB".AtLoadPosition := "Tag__639094376039046365";
               "FB_SortingHeightAdv_DB".AtUnloadPosition := "Tag__639094376039205258";
               "FB_SortingHeightAdv_DB".AtFront := "Tag__639094376039205259";
               "FB_SortingHeightAdv_DB".AtRightEntry := "Tag__639094376039205260";
               "FB_SortingHeightAdv_DB".AtLeftEntry := "Tag__639094376039365268";
               "FB_SortingHeightAdv_DB".AtRightExit := "Tag__639094376039365269";
               "FB_SortingHeightAdv_DB".AtLeftExit := "Tag__639094376039365270";
               "FB_SortingHeightAdv_DB".BtnStart := "Tag__639094376039525211";
               "FB_SortingHeightAdv_DB".BtnReset := "Tag__639094376039525212";
               "FB_SortingHeightAdv_DB".BtnStop := "Tag__639094376039525213";
               "FB_SortingHeightAdv_DB".EmergencyStop := "Tag__639094376039685481";
               "FB_SortingHeightAdv_DB".BtnAuto := "Tag__639094376039685482";
               // â”€â”€ Execute FB â”€â”€
               "FB_SortingHeightAdv_DB"();
               // â”€â”€ Actuators (outputs) â”€â”€
               "Tag__639094376037924724" := "FB_SortingHeightAdv_DB".FeederConveyor;
               "Tag__639094376038085904" := "FB_SortingHeightAdv_DB".EntryConveyor;
               "Tag__639094376038085905" := "FB_SortingHeightAdv_DB".LoadAct;
               "Tag__639094376038405653" := "FB_SortingHeightAdv_DB".UnloadAct;
               "Tag__639094376038565707" := "FB_SortingHeightAdv_DB".TurnAct;
               "Tag__639094376038565708" := "FB_SortingHeightAdv_DB".LeftConveyor;
               "Tag__639094376039846410" := "FB_SortingHeightAdv_DB".RightConveyor;
               "Tag__639094376040005546" := "FB_SortingHeightAdv_DB".GreenIndicator;
               "Tag__639094376038565709" := "FB_SortingHeightAdv_DB".YellowIndicator;
               "Tag__639094376040005547" := "FB_SortingHeightAdv_DB".RedIndicator;
               "Tag__639094376040005548" := "FB_SortingHeightAdv_DB".StartLight;
               "Tag__639094376040163908" := "FB_SortingHeightAdv_DB".ResetLight;
               "Tag__639094376040163909" := "FB_SortingHeightAdv_DB".StopLight;
               "Tag__639094376040963045" := DINT_TO_DWORD("FB_SortingHeightAdv_DB".CounterOut);

           19: // Scene 19: Sorting Height Basic (DB21) â€” 14 inputs, 10 BOOL + 1 DINT outputs
               // â”€â”€ Sensors (inputs) â”€â”€
               // NOTE: Sensors use %I10.x instead of %I0.x to avoid conflict
               // with the PLC's built-in physical digital input module at %IB0.
               "FB_SortingHeightBasic_DB".HighSensor := "Tag__639094376038885860";
               "FB_SortingHeightBasic_DB".LowSensor := "Tag__639094376038885861";
               "FB_SortingHeightBasic_DB".PalletSensor := "Tag__639094376039046363";
               "FB_SortingHeightBasic_DB".Loaded := "Tag__639094376039046364";
               "FB_SortingHeightBasic_DB".AtLeftEntry := "Tag__639094376039046365";
               "FB_SortingHeightBasic_DB".AtLeftExit := "Tag__639094376039205258";
               "FB_SortingHeightBasic_DB".AtRightEntry := "Tag__639094376039205259";
               "FB_SortingHeightBasic_DB".AtRightExit := "Tag__639094376039205260";
               "FB_SortingHeightBasic_DB".BtnStart := "Tag__639094376039365268";
               "FB_SortingHeightBasic_DB".BtnReset := "Tag__639094376039365269";
               "FB_SortingHeightBasic_DB".BtnStop := "Tag__639094376039365270";
               "FB_SortingHeightBasic_DB".EmergencyStop := "Tag__639094376039525211";
               "FB_SortingHeightBasic_DB".BtnAuto := "Tag__639094376039525212";

               "FB_SortingHeightBasic_DB"();

               // â”€â”€ Actuators (outputs) â”€â”€
               "Tag__639094376037924724" := "FB_SortingHeightBasic_DB".ConveyorEntry;
               "Tag__639094376038085904" := "FB_SortingHeightBasic_DB".LoadAct;
               "Tag__639094376038085905" := "FB_SortingHeightBasic_DB".UnloadAct;
               "Tag__639094376038405653" := "FB_SortingHeightBasic_DB".TransfLeft;
               "Tag__639094376038565707" := "FB_SortingHeightBasic_DB".TransfRight;
               "Tag__639094376038565708" := "FB_SortingHeightBasic_DB".ConveyorLeft;
               "Tag__639094376039846410" := "FB_SortingHeightBasic_DB".ConveyorRight;
               "Tag__639094376040005546" := "FB_SortingHeightBasic_DB".StartLight;
               "Tag__639094376038565709" := "FB_SortingHeightBasic_DB".ResetLight;
               "Tag__639094376040005547" := "FB_SortingHeightBasic_DB".StopLight;
               // DINT output for counter display
               "Tag__639094376040963045" := DINT_TO_DWORD("FB_SortingHeightBasic_DB".CounterOut);

           20: // Scene 20: Sorting by Weight (DB22)
               // 14 Bool inputs across %IB10 and %IB11
               "FB_SortingWeight_DB".AtScaleEntry := "Tag__639094376038885860";
               "FB_SortingWeight_DB".AtScale := "Tag__639094376038885861";
               "FB_SortingWeight_DB".AtScaleExit := "Tag__639094376039046363";
               "FB_SortingWeight_DB".AtLeftEntry := "Tag__639094376039046364";
               "FB_SortingWeight_DB".AtExitLeft := "Tag__639094376039046365";
               "FB_SortingWeight_DB".AtForwardEntry := "Tag__639094376039205258";
               "FB_SortingWeight_DB".AtExitFront := "Tag__639094376039205259";
               "FB_SortingWeight_DB".AtRightEntry := "Tag__639094376039205260";
               "FB_SortingWeight_DB".AtExitRight := "Tag__639094376039365268";
               "FB_SortingWeight_DB".BtnStart := "Tag__639094376039365269";
               "FB_SortingWeight_DB".BtnReset := "Tag__639094376039365270";
               "FB_SortingWeight_DB".BtnStop := "Tag__639094376039525211";
               "FB_SortingWeight_DB".BtnAuto := "Tag__639094376039525212";
               "FB_SortingWeight_DB".FIO_Running := "Tag__639094376039525213";
               // Analog: scale weight
               "FB_SortingWeight_DB".Weight := DWORD_TO_REAL("Tag__639094376042076147");
               // Run FB
               "FB_SortingWeight_DB"();
               // 12 Bool outputs
               "Tag__639094376037924724" := "FB_SortingWeight_DB".EntryConveyor;
               "Tag__639094376038085904" := "FB_SortingWeight_DB".LoadScale;
               "Tag__639094376038085905" := "FB_SortingWeight_DB".SendLeft;
               "Tag__639094376038405653" := "FB_SortingWeight_DB".LeftConveyor;
               "Tag__639094376038565707" := "FB_SortingWeight_DB".SendRight;
               "Tag__639094376038565708" := "FB_SortingWeight_DB".RightConveyor;
               "Tag__639094376039846410" := "FB_SortingWeight_DB".SendForward;
               "Tag__639094376040005546" := "FB_SortingWeight_DB".FrontConveyor;
               "Tag__639094376038565709" := "FB_SortingWeight_DB".StartLight;
               "Tag__639094376040005547" := "FB_SortingWeight_DB".ResetLight;
               "Tag__639094376040005548" := "FB_SortingWeight_DB".StopLight;
               // 4 DINT outputs (counts + weight display)
               "Tag__639094376040963045" := DINT_TO_DWORD("FB_SortingWeight_DB".LeftCount);
               "Tag__639094376042315926" := DINT_TO_DWORD("FB_SortingWeight_DB".ForwardCount);
               "Tag__639094376042397245" := DINT_TO_DWORD("FB_SortingWeight_DB".RightCount);
               "Tag__639094376042397246" := DINT_TO_DWORD("FB_SortingWeight_DB".WeightDisplay);

           21: // Scene 21: Sorting Station (DB23)
               // Sensors â€” remapped to %I10.x (avoid built-in DI module)
               "FB_SortingStation_DB".ItemAtEntry := "Tag__639094376038885860";
               "FB_SortingStation_DB".AtDiverter := "Tag__639094376038885861";
               "FB_SortingStation_DB".AtExitGreen := "Tag__639094376039046363";
               "FB_SortingStation_DB".AtExitBlue := "Tag__639094376039046364";
               "FB_SortingStation_DB"();
               "Tag__639094376037924724" := "FB_SortingStation_DB".ConveyorIn;
               "Tag__639094376038085904" := "FB_SortingStation_DB".ConveyorGreen;
               "Tag__639094376038085905" := "FB_SortingStation_DB".ConveyorBlue;
               "Tag__639094376038405653" := "FB_SortingStation_DB".Diverter;
               "Tag__639094376038565707" := "FB_SortingStation_DB".Emitter;
               "Tag__639094376038565708" := "FB_SortingStation_DB".RemoverGreen;
               "Tag__639094376038565709" := "FB_SortingStation_DB".RemoverBlue;

       END_CASE;
END_ORGANIZATION_BLOCK